Omron CX-Programmer project NewProject (CX-Programmer 9.03)

# PLC CLP: CJ1M CPU11
I/O table (CPU CJ1M-CPU11): rack 0 slot 0 CJ1W-ETN21(ETN11Mode); rack 0 slot 1 CJ1W-ID211; rack 0 slot 2 CJ1W-OD211; rack 0 slot 3 CJ1W-ID211; rack 0 slot 4 CJ1W-OD211; rack 0 slot 5 CJ1W-ID211; rack 0 slot 6 CJ1W-OD232

## Global symbols (name address type ; comment)
AS_RS_Ativado 5.02 BOOL
AS_RS_Eixo_X_Ctrg 5.04 BOOL
AS_RS_Eixo_X_D0 5.05 BOOL
AS_RS_Eixo_X_D1 5.06 BOOL
AS_RS_Eixo_X_D2 5.07 BOOL
AS_RS_Eixo_X_D3 5.08 BOOL
AS_RS_Eixo_X_To_Home 5.03 BOOL
AS_RS_Eixo_Y_Ctrg 5.10 BOOL
AS_RS_Eixo_Y_D0 5.11 BOOL
AS_RS_Eixo_Y_D1 5.12 BOOL
AS_RS_Eixo_Y_D2 5.13 BOOL
AS_RS_Eixo_Y_D3 5.14 BOOL
AS_RS_Eixo_Y_To_Home 5.09 BOOL
AS_RS_Eixo_Z_Ctrg 6.00 BOOL
AS_RS_Eixo_Z_D0 6.01 BOOL
AS_RS_Eixo_Z_D1 6.02 BOOL
AS_RS_Eixo_Z_D2 6.03 BOOL
AS_RS_Eixo_Z_D3 6.04 BOOL
AS_RS_Eixo_Z_To_Home 5.15 BOOL
AS_RS_Home_X_Completo 4.05 BOOL
AS_RS_Home_Y_Completo 4.07 BOOL
AS_RS_Home_Z_Completo 4.09 BOOL
AS_RS_Pos_X_Completa 4.04 BOOL
AS_RS_Pos_Y_Completa 4.06 BOOL
AS_RS_Pos_Z_Completa 4.08 BOOL
AUX_CTRG W10.02 BOOL
AUX_X_OK W10.05 BOOL
AUX_X_OK_DESCIDA W16.00 BOOL
AUX_Y_OK W10.07 BOOL
AUX_Z_OK W10.06 BOOL
AUX_Z_OK_DESCIDA W16.01 BOOL
CONF_Z W11.05 BOOL
Confirmacao W4.00 BOOL
Eletroval1 1.06 BOOL
Eletroval2 1.07 BOOL
Eletroval3 1.08 BOOL
Eletroval4 1.09 BOOL
Elevar_Z W15.00 BOOL
Esteira1 1.00 BOOL
Esteira2 1.01 BOOL
Esteira3 1.02 BOOL
Esteira4 1.03 BOOL
Etapa BOOL
Etapa0 W0.00 BOOL
Etapa1 W0.01 BOOL
Etapa10 W1.02 BOOL
Etapa11 W1.03 BOOL
Etapa2 W0.02 BOOL
Etapa3 W0.03 BOOL
Etapa4 W0.04 BOOL
Etapa5 W0.05 BOOL
Etapa6 W0.06 BOOL
Etapa7 W0.07 BOOL
Etapa8 W1.00 BOOL
Etapa9 W1.01 BOOL
Home_X_Completo 4.05 BOOL
Home_Y_Completo 4.07 BOOL
Home_Z_Completo 4.09 BOOL
Pos_X_Completa 4.04 BOOL
Pos_Y_Completa 4.06 BOOL
Pos_Z_Completa 4.08 BOOL
Sensor1 0.00 BOOL
Sensor2 0.01 BOOL
Sensor3 0.02 BOOL
Sensor4 0.03 BOOL
X_CTRG 5.04 BOOL
X_D0 5.05 BOOL
X_D1 5.06 BOOL
X_D2 5.07 BOOL
X_D3 5.08 BOOL
X_To_Home 5.03 BOOL
Y_CTRG 5.10 BOOL
Y_D0 5.11 BOOL
Y_D1 5.12 BOOL
Y_D2 5.13 BOOL
Y_D3 5.14 BOOL
Y_To_Home 5.09 BOOL
Z_CTRG 6.00 BOOL
Z_D0 6.01 BOOL
Z_D1 6.02 BOOL
Z_D2 6.03 BOOL
Z_D3 6.04 BOOL
Z_To_Home 5.15 BOOL

## Program NewProgram1 (cyclic task 0)
Local symbols
AS_RS_Ativado 5.02 BOOL
AUX_CTRG W10.02 BOOL
AUX_ROBO_OK W50.00 BOOL
AUX_VISAO_OK W50.01 BOOL
AUX_X_OK W10.05 BOOL
AUX_Y_OK W10.07 BOOL
AUX_Z_OK W10.06 BOOL
Confirmacao W4.00 BOOL
Eletroval1 1.06 BOOL
Eletroval2 1.07 BOOL
Eletroval3 1.08 BOOL
Eletroval4 1.09 BOOL
Elevar_Z W15.00 BOOL
Esteira1 1.00 BOOL
Esteira2 1.01 BOOL
Esteira3 1.02 BOOL
Esteira4 1.03 BOOL
Etapa BOOL
Etapa0 W0.00 BOOL
Etapa1 W0.01 BOOL
Etapa10 W1.02 BOOL
Etapa11 W1.03 BOOL
Etapa12 W1.04 BOOL
Etapa13 W1.05 BOOL
Etapa14 W1.06 BOOL
Etapa15 W1.07 BOOL
Etapa16 W2.00 BOOL
Etapa17 W2.01 BOOL
Etapa18 W2.02 BOOL
Etapa19 W2.03 BOOL
Etapa2 W0.02 BOOL
Etapa20 W2.04 BOOL
Etapa21 W2.05 BOOL
Etapa22 W2.06 BOOL
Etapa23 W2.07 BOOL
Etapa24 W3.01 BOOL
Etapa25 W3.02 BOOL
Etapa26 W3.03 BOOL
Etapa27 W3.04 BOOL
Etapa28 W3.05 BOOL
Etapa29 W3.06 BOOL
Etapa3 W0.03 BOOL
Etapa30 W3.07 BOOL
Etapa4 W0.04 BOOL
Etapa5 W0.05 BOOL
Etapa6 W0.06 BOOL
Etapa7 W0.07 BOOL
Etapa8 W1.00 BOOL
Etapa9 W1.01 BOOL
FLAG_ROBO W50.02 BOOL
Home_X_Completo 4.05 BOOL
Home_Y_Completo 4.07 BOOL
Home_Z_Completo 4.09 BOOL
MAO_PEGAR_ARMAZEM 6.08 BOOL
MAO_PEGAR_ESTEIRA 6.09 BOOL
Pos_X_Completa 4.04 BOOL
Pos_Y_Completa 4.06 BOOL
Pos_Z_Completa 4.08 BOOL
Sensor1 0.00 BOOL
Sensor2 0.01 BOOL
Sensor3 0.02 BOOL
Sensor4 0.03 BOOL
WORD_X W35 WORD
WORD_Z W40 WORD
XD0 BOOL
X_CTRG 5.04 BOOL
X_D0 5.05 BOOL
X_D1 5.06 BOOL
X_D2 5.07 BOOL
X_D3 5.08 BOOL
X_To_Home 5.03 BOOL
Y_CTRG 5.10 BOOL
Y_D0 5.11 BOOL
Y_D1 5.12 BOOL
Y_D2 5.13 BOOL
Y_D3 5.14 BOOL
Y_To_Home 5.09 BOOL
Z_CTRG 6.00 BOOL
Z_D0 6.01 BOOL
Z_D1 6.02 BOOL
Z_D2 6.03 BOOL
Z_D3 6.04 BOOL
Z_To_Home 5.15 BOOL

### Section Armazem_esteiras

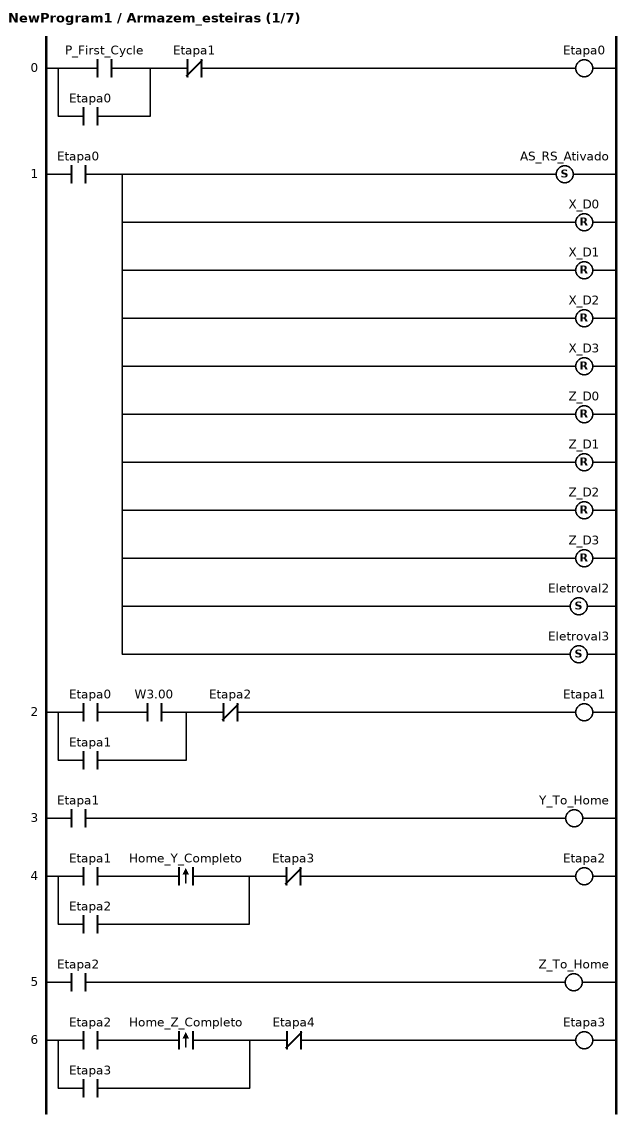
; rung 0
LD P_First_Cycle
OR Etapa0
ANDNOT Etapa1
OUT Etapa0
; rung 1
LD Etapa0
SET AS_RS_Ativado
RSET X_D0
RSET X_D1
RSET X_D2
RSET X_D3
RSET Z_D0
RSET Z_D1
RSET Z_D2
RSET Z_D3
SET Eletroval2
SET Eletroval3
; rung 2
LD Etapa0
AND W3.00
OR Etapa1
ANDNOT Etapa2
OUT Etapa1
; rung 3
LD Etapa1
OUT Y_To_Home
; rung 4
LD Etapa1
@AND Home_Y_Completo
OR Etapa2
ANDNOT Etapa3
OUT Etapa2
; rung 5
LD Etapa2
OUT Z_To_Home
; rung 6
LD Etapa2
@AND Home_Z_Completo
OR Etapa3
ANDNOT Etapa4
OUT Etapa3

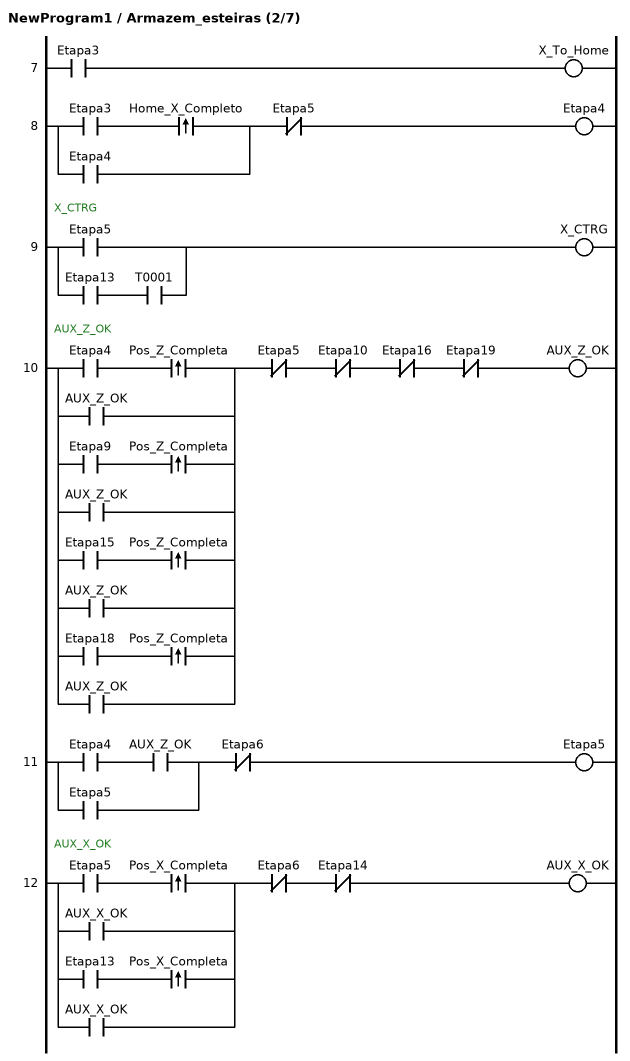
; rung 7
LD Etapa3
OUT X_To_Home
; rung 8
LD Etapa3
@AND Home_X_Completo
OR Etapa4
ANDNOT Etapa5
OUT Etapa4
; rung 9: X_CTRG
LD Etapa5
LD Etapa13
AND T0001
ORLD
OUT X_CTRG
; rung 10: AUX_Z_OK
LD Etapa4
@AND Pos_Z_Completa
OR AUX_Z_OK
LD Etapa9
@AND Pos_Z_Completa
ORLD
OR AUX_Z_OK
LD Etapa15
@AND Pos_Z_Completa
ORLD
OR AUX_Z_OK
LD Etapa18
@AND Pos_Z_Completa
ORLD
OR AUX_Z_OK
ANDNOT Etapa5
ANDNOT Etapa10
ANDNOT Etapa16
ANDNOT Etapa19
OUT AUX_Z_OK
; rung 11
LD Etapa4
AND AUX_Z_OK
OR Etapa5
ANDNOT Etapa6
OUT Etapa5
; rung 12: AUX_X_OK
LD Etapa5
@AND Pos_X_Completa
OR AUX_X_OK
LD Etapa13
@AND Pos_X_Completa
ORLD
OR AUX_X_OK
ANDNOT Etapa6
ANDNOT Etapa14
OUT AUX_X_OK

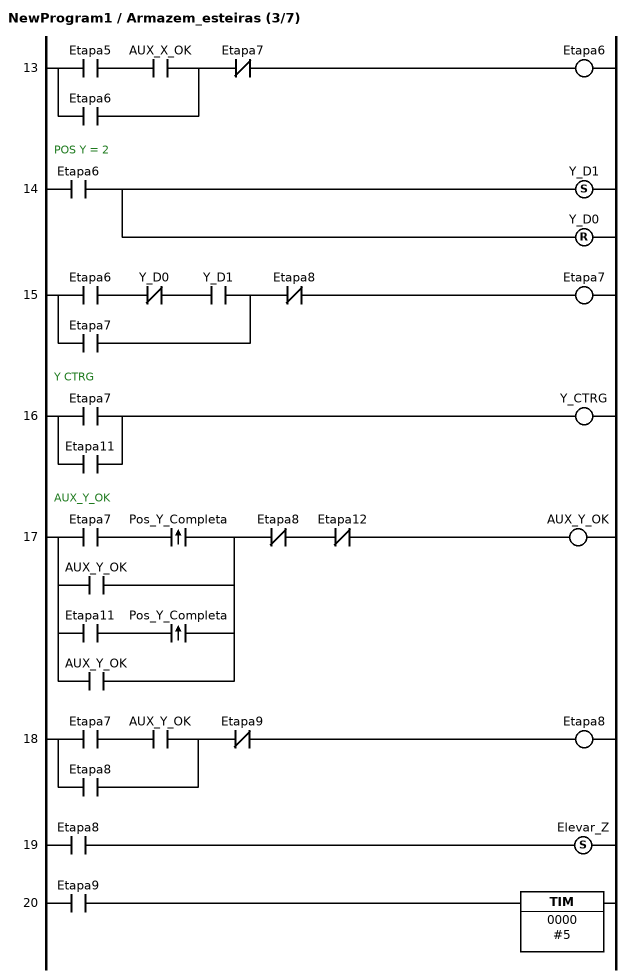
; rung 13
LD Etapa5
AND AUX_X_OK
OR Etapa6
ANDNOT Etapa7
OUT Etapa6
; rung 14: POS Y = 2
LD Etapa6
SET Y_D1
RSET Y_D0
; rung 15
LD Etapa6
ANDNOT Y_D0
AND Y_D1
OR Etapa7
ANDNOT Etapa8
OUT Etapa7
; rung 16: Y CTRG
LD Etapa7
OR Etapa11
OUT Y_CTRG
; rung 17: AUX_Y_OK
LD Etapa7
@AND Pos_Y_Completa
OR AUX_Y_OK
LD Etapa11
@AND Pos_Y_Completa
ORLD
OR AUX_Y_OK
ANDNOT Etapa8
ANDNOT Etapa12
OUT AUX_Y_OK
; rung 18
LD Etapa7
AND AUX_Y_OK
OR Etapa8
ANDNOT Etapa9
OUT Etapa8
; rung 19
LD Etapa8
SET Elevar_Z
; rung 20
LD Etapa9
TIM 0000 #5

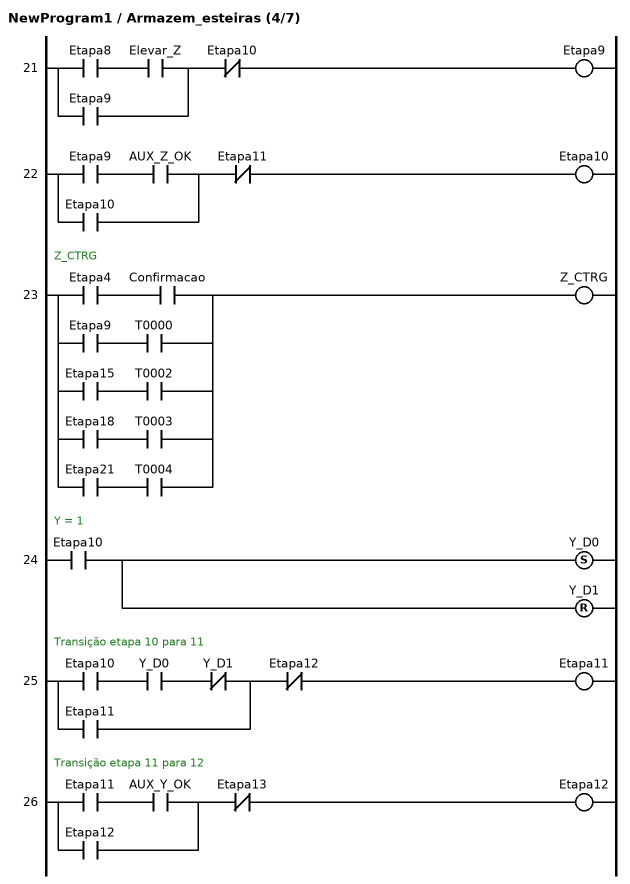
; rung 21
LD Etapa8
AND Elevar_Z
OR Etapa9
ANDNOT Etapa10
OUT Etapa9
; rung 22
LD Etapa9
AND AUX_Z_OK
OR Etapa10
ANDNOT Etapa11
OUT Etapa10
; rung 23: Z_CTRG
LD Etapa4
AND Confirmacao
LD Etapa9
AND T0000
ORLD
LD Etapa15
AND T0002
ORLD
LD Etapa18
AND T0003
ORLD
LD Etapa21
AND T0004
ORLD
OUT Z_CTRG
; rung 24: Y = 1
LD Etapa10
SET Y_D0
RSET Y_D1
; rung 25: Transição etapa 10 para 11
LD Etapa10
AND Y_D0
ANDNOT Y_D1
OR Etapa11
ANDNOT Etapa12
OUT Etapa11
; rung 26: Transição etapa 11 para 12
LD Etapa11
AND AUX_Y_OK
OR Etapa12
ANDNOT Etapa13
OUT Etapa12

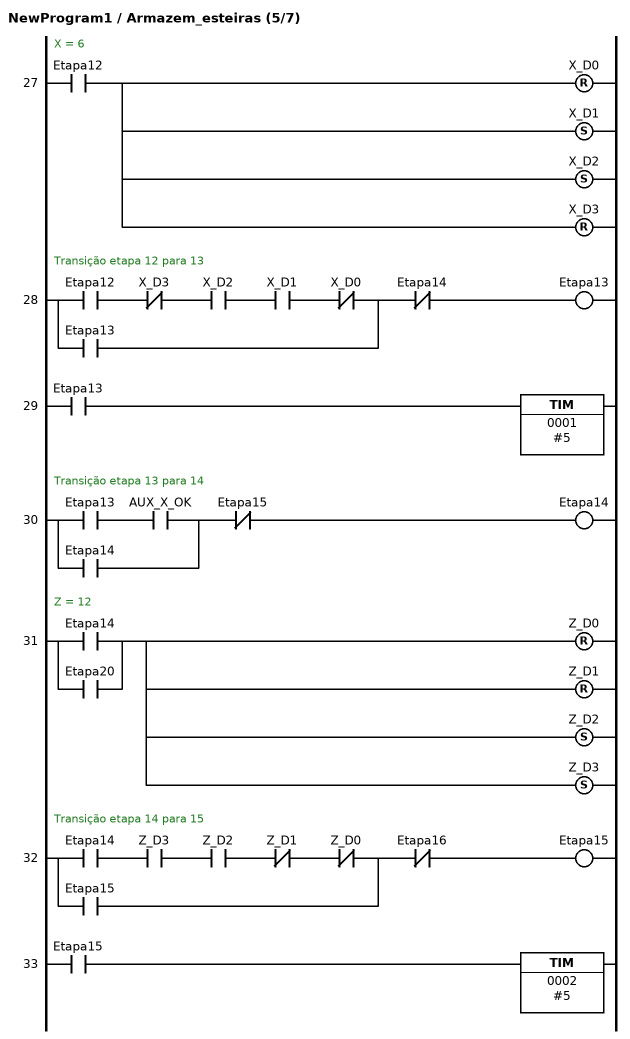
; rung 27: X = 6
LD Etapa12
RSET X_D0
SET X_D1
SET X_D2
RSET X_D3
; rung 28: Transição etapa 12 para 13
LD Etapa12
ANDNOT X_D3
AND X_D2
AND X_D1
ANDNOT X_D0
OR Etapa13
ANDNOT Etapa14
OUT Etapa13
; rung 29
LD Etapa13
TIM 0001 #5
; rung 30: Transição etapa 13 para 14
LD Etapa13
AND AUX_X_OK
OR Etapa14
ANDNOT Etapa15
OUT Etapa14
; rung 31: Z = 12
LD Etapa14
OR Etapa20
RSET Z_D0
RSET Z_D1
SET Z_D2
SET Z_D3
; rung 32: Transição etapa 14 para 15
LD Etapa14
AND Z_D3
AND Z_D2
ANDNOT Z_D1
ANDNOT Z_D0
OR Etapa15
ANDNOT Etapa16
OUT Etapa15
; rung 33
LD Etapa15
TIM 0002 #5

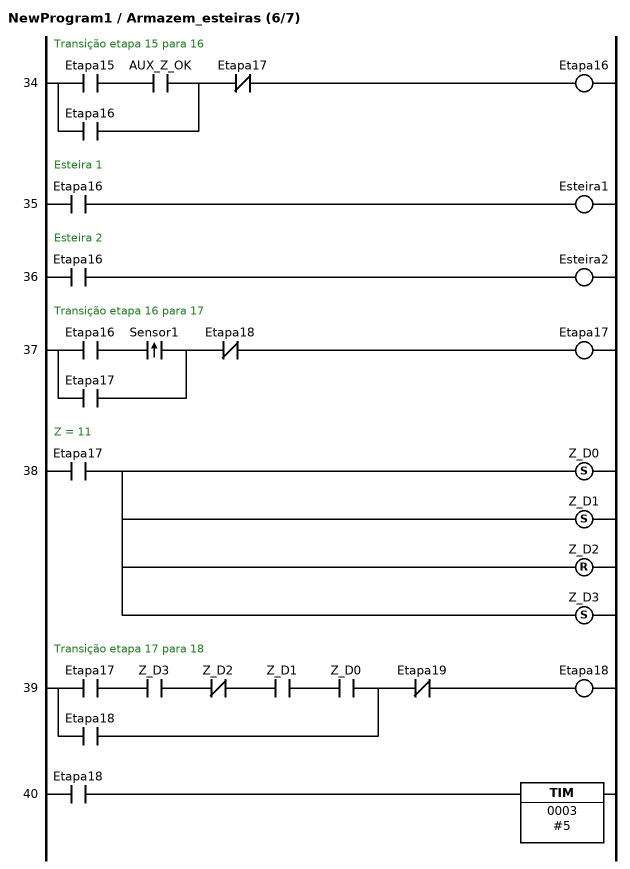
; rung 34: Transição etapa 15 para 16
LD Etapa15
AND AUX_Z_OK
OR Etapa16
ANDNOT Etapa17
OUT Etapa16
; rung 35: Esteira 1
LD Etapa16
OUT Esteira1
; rung 36: Esteira 2
LD Etapa16
OUT Esteira2
; rung 37: Transição etapa 16 para 17
LD Etapa16
@AND Sensor1
OR Etapa17
ANDNOT Etapa18
OUT Etapa17
; rung 38: Z = 11
LD Etapa17
SET Z_D0
SET Z_D1
RSET Z_D2
SET Z_D3
; rung 39: Transição etapa 17 para 18
LD Etapa17
AND Z_D3
ANDNOT Z_D2
AND Z_D1
AND Z_D0
OR Etapa18
ANDNOT Etapa19
OUT Etapa18
; rung 40
LD Etapa18
TIM 0003 #5

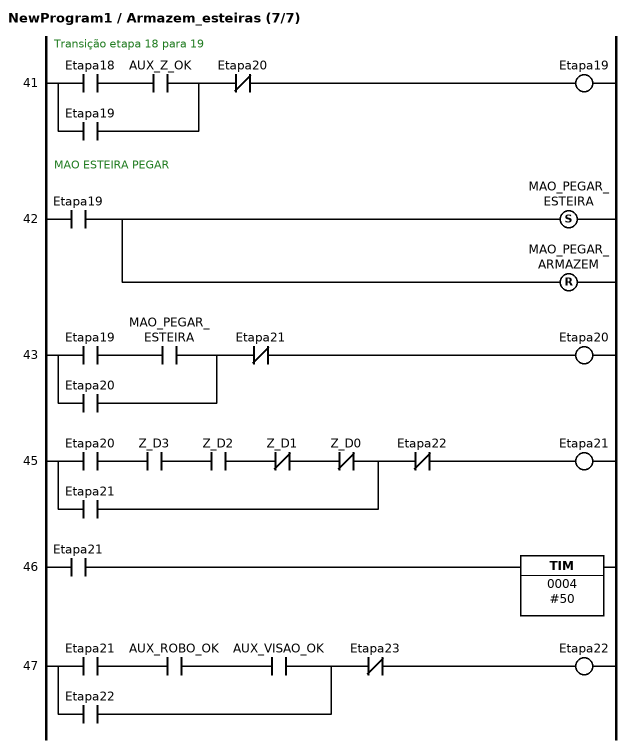
; rung 41: Transição etapa 18 para 19
LD Etapa18
AND AUX_Z_OK
OR Etapa19
ANDNOT Etapa20
OUT Etapa19
; rung 42: MAO ESTEIRA PEGAR
LD Etapa19
SET MAO_PEGAR_ESTEIRA
RSET MAO_PEGAR_ARMAZEM
; rung 43
LD Etapa19
AND MAO_PEGAR_ESTEIRA
OR Etapa20
ANDNOT Etapa21
OUT Etapa20
; rung 44: MAO ARMAZEM PEGAR
; rung 45
LD Etapa20
AND Z_D3
AND Z_D2
ANDNOT Z_D1
ANDNOT Z_D0
OR Etapa21
ANDNOT Etapa22
OUT Etapa21
; rung 46
LD Etapa21
TIM 0004 #50
; rung 47
LD Etapa21
AND AUX_ROBO_OK
AND AUX_VISAO_OK
OR Etapa22
ANDNOT Etapa23
OUT Etapa22

### Section Transitions

### Section Robo

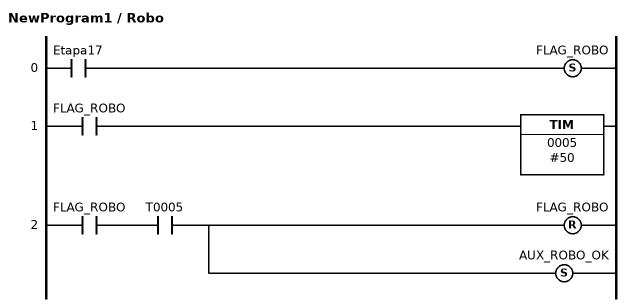
; rung 0
LD Etapa17
SET FLAG_ROBO
; rung 1
LD FLAG_ROBO
TIM 0005 #50
; rung 2
LD FLAG_ROBO
AND T0005
RSET FLAG_ROBO
SET AUX_ROBO_OK

### Section Visao

### Section END
; rung 0
END(001)